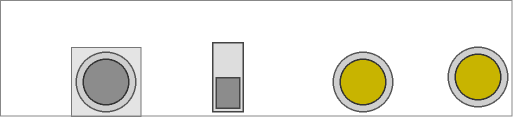
VISUALIZATION Visualization  // 513x117
    PushSwitch (71,47 70x70), variable: GVL.BoutonVirtuel, behaviour: TOGGLE, style: Switch-PushSwitch-Gray
    Lamp1 (443,42 70x70), variable: GVL.LumiereDroite, style: Lamp-Lamp1-Yellow
    Lamp1 (328,47 70x70), variable: GVL.LumiereGauche, style: Lamp-Lamp1-Yellow
    DipSwitch (193,42 70x70), variable: GVL.BoutonSelecteur, behaviour: TOGGLE, style: Switch-DipSwitch-Gray
END_VISUALIZATION

(* stored: Version 1.1.0.1, ProductVersion 3.1.4024.16
   Visu Visualization: Id {7f40df0f-979c-4df7-baa7-77fd2fc40876} *)
